ABB RAPID module: MainModule.mod

MODULE MainModule
    !***********************************************************
    ! @file MainModule.mod
    ! @brief Glavni modul aplikacije za automatsko paletiranje.
    !
    ! @details
    ! Ovaj modul sadrzi glavni tok izvrsavanja programa.
    ! Program radi ciklicno i u svakom ciklusu izvrsava sledece
    ! korake:
    !
    ! 1. Resetovanje aktivnog rasporeda palete.
    ! 2. Cekanje da korisnik unese raspored preko ScreenMaker HMI-ja.
    ! 3. Odlazak robota u neutralnu poziciju kako ne bi zaklanjao
    !    vidno polje kamere.
    ! 4. Simulacija ocitavanja kamere.
    ! 5. Azuriranje aktivnog WorkObject-a palete na osnovu
    !    vrednosti koje vrati kamera.
    ! 6. Cekanje dozvole operatora preko digitalnog ulaza
    !    StartProces.
    ! 7. Izvrsavanje pick/place procesa paletiranja.
    ! 8. Povratak robota u home poziciju i priprema za novi ciklus.
    !
    ! U ovom modulu se ne nalaze pojedinacne pick/place putanje,
    ! vec se one pozivaju preko procedura iz modula PalletLogic,
    ! PickPaths i PlacePaths.
    !***********************************************************



    !***********************************************************
    ! @brief Neutralna pozicija robota za ocitavanje kamere.
    !
    ! @details
    ! Robtarget predstavlja poziciju u koju se robot pomera pre
    ! simulacije kamere. U ovoj poziciji se pretpostavlja da robot
    ! ne zaklanja vidno polje kamere postavljene iznad postolja.
    !***********************************************************
    CONST robtarget pCameraClear:=[[-19.230864356,-323.825304784,292.236710827],[0.082629296,0.722256662,0.681057326,-0.087627807],[-2,-1,-1,0],[9E+09,9E+09,9E+09,9E+09,9E+09,9E+09]];


    !***********************************************************
    ! @brief Home pozicija robota.
    !
    ! @details
    ! Robtarget predstavlja bezbednu/pocetnu poziciju robota.
    ! Robot se u ovu poziciju vraca nakon zavrsetka ciklusa
    ! paletiranja.
    !***********************************************************
    CONST robtarget pHome:=[[477.110336645,-0.2,528.9],[0.5,0,0.866025404,0],[0,0,0,0],[9E+09,9E+09,9E+09,9E+09,9E+09,9E+09]];


    !***********************************************************
    ! @brief Cekanje da korisnik unese validan raspored palete.
    !
    ! @details
    ! Procedura periodicno poziva HMI_Handler(), koji obradjuje
    ! zahteve sa ScreenMaker HMI-ja. Korisnik preko HMI-ja unosi
    ! boju kockice i poziciju na paleti, a zatim dodaje unos u
    ! raspored.
    !
    ! Procedura ne dozvoljava nastavak programa dok korisnik ne
    ! potvrdi raspored i dok raspored ne ispuni uslov da se svaka
    ! boja nalazi na barem jednoj poziciji palete.
    !
    ! Ako raspored nije validan, korisniku se ispisuje statusna
    ! poruka i program nastavlja da ceka novi unos/potvrdu.
    !***********************************************************
    PROC WaitForValidPattern()
        VAR bool patternReady;

        patternReady := FALSE;
        hmiStartReq := FALSE;

        SetStatus "Unesi raspored kockica preko HMI-ja.";

        WHILE NOT patternReady DO

            WHILE NOT hmiStartReq DO
                HMI_Handler;
                WaitTime 0.1;
            ENDWHILE

            ! Obradi eventualni poslednji klik na ADD/RESET pre starta
            HMI_Handler;

            IF IsPatternValid() THEN
                patternReady := TRUE;
                hmiStartReq := FALSE;
                SetStatus "Raspored je validan.";
            ELSE
                SetStatus "Greska: svaka boja mora biti uneta bar jednom.";
                hmiStartReq := FALSE;
            ENDIF
        ENDWHILE
    ENDPROC


    !***********************************************************
    ! @brief Glavni program aplikacije.
    !
    ! @details
    ! Glavni program izvrsava kompletan ciklus paletiranja.
    ! Na pocetku svakog ciklusa aktivni WorkObject palete
    ! wobjPaleta se vraca na nominalnu vrednost wobjPaletaNominal.
    !
    ! Nakon unosa i validacije rasporeda, robot odlazi u poziciju
    ! pCameraClear, zatim se poziva funkcija SimulateCameraReading()
    ! koja simulira ocitavanje kamere. Dobijene vrednosti X, Y i Rz
    ! koriste se za korekciju aktivnog koordinatnog sistema palete.
    !
    ! Program zatim ceka digitalni ulaz StartProces. Kada operator
    ! da dozvolu, poziva se Palletize(), cime se izvrsava kompletan
    ! pick/place proces prema unetom rasporedu.
    !
    ! Nakon zavrsetka paletiranja robot se vraca u home poziciju i
    ! ceka da se StartProces vrati na nulu, kako novi ciklus ne bi
    ! krenuo automatski.
    !***********************************************************
PROC main()
    VAR camerapos detected;

    ! Inicijalizacija semena za pseudo-random simulaciju kamere.
    InitRandomSeed;

    WHILE TRUE DO
        ! Pre svakog ciklusa aktivna paleta se vraca na nominalni,
        ! rucno nauceni polozaj. Time se sprecava akumulacija offseta
        ! iz prethodnih ciklusa.
        wobjPaleta := wobjPaletaNominal;

        ! Brisanje prethodnog rasporeda i priprema za novi unos.
        ResetPattern;
        SetStatus "Novi ciklus: unesi raspored.";

        ! Cekanje da korisnik preko HMI-ja unese validan raspored.
        ! Program se ne nastavlja dok svaka boja nije uneta bar jednom.
        WaitForValidPattern;

        ! Robot se sklanja u poziciju u kojoj ne zaklanja kameru.
        SetStatus "Robot se sklanja iz vidnog polja kamere.";
        Path_CameraClear;

        ! Simulirana kamera vraca X, Y i Rz offset palete u odnosu
        ! na nominalni polozaj. Za stabilnu simulaciju koristi se mali
        ! opseg pomeraja i rotacije.
        detected := SimulateCameraReading(-20, 20, -20, 20, -5, 5);

        TPWrite "Camera X: " + ValToStr(detected.x);
        TPWrite "Camera Y: " + ValToStr(detected.y);
        TPWrite "Camera Rz: " + ValToStr(detected.rz);

        SetStatus "Kamera: X=" + ValToStr(detected.x) +
                  " Y=" + ValToStr(detected.y) +
                  " Rz=" + ValToStr(detected.rz);

        ! Na osnovu vrednosti kamere azurira se aktivni WorkObject
        ! palete. Sve place tacke koriste wobjPaleta, pa se automatski
        ! pomeraju zajedno sa paletom.
        UpdatePalletWObjOffset detected;

        ! Nakon unosa rasporeda i ocitavanja kamere, operator mora
        ! dati dozvolu za pocetak paletiranja preko digitalnog ulaza.
        SetStatus "Cekam dozvolu operatora: StartProces.";
        WaitDI StartProces, 1;

        ! Izvrsavanje kompletnog pick/place procesa prema unetom rasporedu.
        SetStatus "Paletiranje u toku.";
        Palletize;

        SetStatus "Paletiranje zavrseno.";

        ! Povratak robota u home poziciju nakon zavrsenog ciklusa.
        Path_HomePosition;

        ! Aktivna paleta se vraca na nominalnu vrednost nakon ciklusa,
        ! kako bi sledeci ciklus poceo iz poznatog stanja.
        wobjPaleta := wobjPaletaNominal;

        ! Cekanje da operator otpusti StartProces signal. Ovo sprecava
        ! automatski ulazak u sledeci ciklus dok je signal jos uvek aktivan.
        WaitDI StartProces, 0;
    ENDWHILE
ENDPROC


    !***********************************************************
    ! @brief Pomera robota u poziciju u kojoj ne zaklanja kameru.
    !
    ! @details
    ! Procedura izvrsava MoveJ kretanje do targeta pCameraClear.
    ! Koristi se pre simulacije ocitavanja kamere, kako bi se
    ! obezbedilo da robot ne ometa vidno polje kamere.
    !***********************************************************
    PROC Path_CameraClear()
        MoveJ pCameraClear,v1000,fine,Vakuum_Griepr\WObj:=wobj0;
    ENDPROC

    !***********************************************************
    ! @brief Pomera robota u home poziciju.
    !
    ! @details
    ! Procedura izvrsava MoveJ kretanje do targeta pHome.
    ! Koristi se nakon zavrsetka ciklusa paletiranja, kao i za
    ! postavljanje robota u bezbednu/pocetnu poziciju.
    !***********************************************************
    PROC Path_HomePosition()
        MoveJ pHome,v1000,fine,Vakuum_Griepr\WObj:=wobj0;
    ENDPROC


    !***********************************************************
    ! @brief Azurira aktivni WorkObject palete na osnovu kamere.
    !
    ! @details
    ! Procedura prima strukturu camerapos, koja sadrzi vrednosti
    ! x, y i rz dobijene simulacijom kamere.
    !
    ! Vrednosti x i y predstavljaju translacioni pomeraj palete,
    ! dok rz predstavlja rotaciju palete oko Z ose. Na osnovu tih
    ! vrednosti formira se offsetPose.
    !
    ! Aktivni WorkObject wobjPaleta se racuna kao nominalni
    ! WorkObject wobjPaletaNominal pomeren za izracunati offset.
    ! Na taj nacin sve place tacke, koje su definisane lokalno u
    ! odnosu na wobjPaleta, automatski prate pomeraj palete.
    !
    ! @param cam Rezultat simuliranog ocitavanja kamere.
    !***********************************************************
    PROC UpdatePalletWObjOffset(camerapos cam)
        VAR pose offsetPose;

        offsetPose.trans := [cam.x, cam.y, 0];
        offsetPose.rot := OrientZYX(cam.rz, 0, 0);

        ! Aktivna paleta = nominalna paleta + offset kamere.
        wobjPaleta.uframe := PoseMult(wobjPaletaNominal.uframe, offsetPose);
        wobjPaleta.oframe := wobjPaletaNominal.oframe;
    ENDPROC
ENDMODULE
